// TwinCAT 3 PLC project tcp_client
// ProgramVersion: 3.1.4024.0
// libraries:
//   Tc2_Standard, * (Beckhoff Automation GmbH)
//   Tc2_System, * (Beckhoff Automation GmbH)
//   Tc2_TcpIp, * (Beckhoff Automation GmbH)
//   Tc3_Module, * (Beckhoff Automation GmbH)
// project tree:
//   GVLs/ SockParam.TcGVL
//   / PlcTask.TcTTO
//   POUs/libSocketClient/ E_SocketCommStateMachine.TcDUT, FB_SocketClientController.TcPOU, FB_MessageQueue.TcPOU, ITF_Receiver.TcIO, ITF_Sender.TcIO, ITF_TaskObserver.TcIO, ST_CommunicationMetaData.TcDUT, ST_CommandContainer.TcDUT
//   POUs/ MAIN.TcPOU
//   POUs/protocols/ FB_SocketClientProtocolBase.TcPOU
//   POUs/protocols/TestProtocol/ FB_TestProtocol.TcPOU, ST_ReceiveDataFormat.TcDUT, ST_SendDataFormat.TcDUT
// real-time tasks:
//   TASK PlcTask: cycle T#10ms, priority 20, ADS port 350

CONFIGURATION tcp_client
    RESOURCE PLC ON TwinCAT3
        TASK PlcTask(INTERVAL := T#10ms, PRIORITY := 20);
        PROGRAM MAIN WITH PlcTask : MAIN;
    END_RESOURCE
END_CONFIGURATION

// ---- POUs/libSocketClient/E_SocketCommStateMachine.TcDUT
{attribute 'qualified_only'}
{attribute 'strict'}
TYPE E_SocketCommStateMachine :
(
	init := 0,
	connect,
	idle,
	send,
	receive,
	disconnect,
	done
);
END_TYPE

// ---- POUs/libSocketClient/ST_CommunicationMetaData.TcDUT
TYPE ST_CommunicationMetaData :
STRUCT
	cbLen	: UDINT;
	pData	: PVOID;
END_STRUCT
END_TYPE

// ---- POUs/libSocketClient/ST_CommandContainer.TcDUT
TYPE ST_CommandContainer :
STRUCT
	sender : ITF_Sender;
	receiver : ITF_receiver;
END_STRUCT
END_TYPE

// ---- POUs/protocols/TestProtocol/ST_ReceiveDataFormat.TcDUT
{attribute 'pack_mode' := '1'}
TYPE ST_ReceiveDataFormat :
STRUCT
   command        : STRING(4);
   seq_number    : ULINT;
   value        : STRING(10240);
END_STRUCT
END_TYPE

// ---- POUs/protocols/TestProtocol/ST_SendDataFormat.TcDUT
{attribute 'pack_mode' := '1'}
TYPE ST_SendDataFormat :
STRUCT
   command        : STRING(4);
   seq_number    : ULINT;
   value        : ULINT;
END_STRUCT
END_TYPE

// ---- GVLs/SockParam.TcGVL
{attribute 'qualified_only'}
VAR_GLOBAL CONSTANT
	MAX_MESSAGE_SIZE : UDINT := 2048;	// 受信処理バッファ最大サイズ
	RECEIVE_BUFFER_SIZE	: UDINT := 20480; // 受信メッセージの組立先のバッファサイズ
END_VAR

// ---- POUs/libSocketClient/ITF_Receiver.TcIO
INTERFACE ITF_Receiver EXTENDS __System.IQueryInterface

METHOD flush : BOOL
VAR_INPUT
END_VAR
END_METHOD

METHOD Parse : BOOL
VAR_INPUT
END_VAR
END_METHOD

PROPERTY received : BOOL
GET
END_GET
END_PROPERTY

METHOD ResetBufferPointer : BOOL
VAR_INPUT
END_VAR
END_METHOD

METHOD SetReceivedData : BOOL
VAR_INPUT
	pData	: PVOID;
	cbLen	: UDINT;
END_VAR
END_METHOD

END_INTERFACE

// ---- POUs/libSocketClient/ITF_Sender.TcIO
INTERFACE ITF_Sender EXTENDS __System.IQueryInterface

PROPERTY SendData : ST_CommunicationMetaData
GET
END_GET
END_PROPERTY

END_INTERFACE

// ---- POUs/libSocketClient/ITF_TaskObserver.TcIO
INTERFACE ITF_TaskObserver EXTENDS __System.IQueryInterface

PROPERTY activity : E_SocketCommStateMachine
GET
END_GET
SET
END_SET
END_PROPERTY

PROPERTY complete : BOOL
GET
END_GET
SET
END_SET
END_PROPERTY

PROPERTY error : BOOL
GET
END_GET
SET
END_SET
END_PROPERTY

PROPERTY error_id : UDINT
GET
END_GET
SET
END_SET
END_PROPERTY

END_INTERFACE

// ---- POUs/MAIN.TcPOU
PROGRAM MAIN
VAR
	protcol : FB_TestProtocol;
	controller : FB_SocketClientController;
	connect : BOOL;
	handle : T_HSOCKET;
	
	// Command execution
	command_interval_timer : TON := (PT := T#1S);
	rand : DRAND;
	busy : BOOL;
	// Receive data
	receive_data : REFERENCE TO ST_ReceiveDataFormat;	
	
END_VAR

IF connect THEN
	handle := controller.connect('127.0.0.1', 9998);
ELSE
	controller.disconnect();
	busy := FALSE;
END_IF

IF handle.handle <> 0 THEN
	command_interval_timer(IN := NOT command_interval_timer.Q);
	IF command_interval_timer.Q AND NOT busy THEN
		rand(Seed := 1);
		protcol.send_data.command := 'SEND';
		protcol.send_data.seq_number := protcol.send_data.seq_number + 1;
		protcol.send_data.value := TO_ULINT(rand.Num * 100000);
		controller.queue.put(protcol, protcol);
		busy := TRUE;
	END_IF
	IF busy AND protcol.complete THEN
		receive_data REF= protcol.receive_data;
		busy := FALSE;
	END_IF
END_IF

controller();

END_PROGRAM

// ---- POUs/protocols/TestProtocol/FB_TestProtocol.TcPOU

FUNCTION_BLOCK FB_TestProtocol EXTENDS FB_SocketClientProtocolBase
VAR_INPUT
	send_data : ST_SendDataFormat;
END_VAR
VAR_OUTPUT
	receive_data : ST_ReceiveDataFormat;
END_VAR
VAR
END_VAR

METHOD Parse : BOOL
IF SIZEOF(receive_data) = MEMCPY(ADR(receive_data), ADR(SUPER^.receive_data_buffer), SIZEOF(receive_data)) THEN
	Parse := TRUE;
END_IF
END_METHOD

PROPERTY received : BOOL
GET
VAR
	specified_size : UDINT;
END_VAR
specified_size := SIZEOF(receive_data);
received := SUPER^.receive_data_size = specified_size;
END_GET
END_PROPERTY

PROPERTY SendData : ST_CommunicationMetaData
GET
SendData.cbLen := SIZEOF(send_data);
SendData.pData := ADR(send_data);
END_GET
END_PROPERTY

END_FUNCTION_BLOCK

// ---- POUs/protocols/FB_SocketClientProtocolBase.TcPOU
FUNCTION_BLOCK ABSTRACT FB_SocketClientProtocolBase IMPLEMENTS ITF_Sender, ITF_Receiver, ITF_TaskObserver
VAR CONSTANT
	MAX_NUM_OF_REQUEST_SECTIONS : UINT := 16;
END_VAR
VAR_OUTPUT
	//ParsedStructVariable : ST_********;
END_VAR
VAR	
	expected_receive_size_min : UDINT := 1; 
	expected_receive_size_max : UDINT := 1024; 
	receive_data_buffer	: ARRAY [0..SockParam.RECEIVE_BUFFER_SIZE - 1] OF BYTE;
	receive_data_size	: UDINT;
	_activity : E_SocketCommStateMachine;
	_error		: BOOL;
	_complete	: BOOL;
	_error_id	: UDINT;
END_VAR

PROPERTY activity : E_SocketCommStateMachine
GET
activity := _activity;
END_GET
SET
_activity := activity;
END_SET
END_PROPERTY

PROPERTY complete : BOOL
GET
complete := _complete;
END_GET
SET
_complete := complete;
END_SET
END_PROPERTY

PROPERTY error : BOOL
GET
error := _error;
END_GET
SET
_error := error;
END_SET
END_PROPERTY

PROPERTY error_id : UDINT
GET
error_id := _error_id;
END_GET
SET
_error_id := error_id;
END_SET
END_PROPERTY

METHOD FB_init : BOOL
VAR_INPUT
	bInitRetains : BOOL; // if TRUE, the retain variables are initialized (warm start / cold start)
	bInCopyCode : BOOL;  // if TRUE, the instance afterwards gets moved into the copy code (online change)
END_VAR
THIS^.flush();
END_METHOD

METHOD flush : BOOL
receive_data_size := 0;
END_METHOD

METHOD Parse : BOOL
END_METHOD

PROPERTY received : BOOL
GET
END_GET
END_PROPERTY

METHOD ResetBufferPointer : BOOL
receive_data_size := 0;
END_METHOD

PROPERTY SendData : ST_CommunicationMetaData
GET
END_GET
END_PROPERTY

METHOD SetReceivedData : BOOL
VAR_INPUT
	pData	: PVOID;
	cbLen	: UDINT;
END_VAR
VAR
	i : UDINT;
END_VAR
IF pData = 0 OR cbLen = 0 THEN
	RETURN;
END_IF

MEMCPY(ADR(receive_data_buffer) + receive_data_size, pData, cbLen);
receive_data_size := receive_data_size + cbLen;
SetReceivedData := TRUE;
END_METHOD

END_FUNCTION_BLOCK

// ---- POUs/libSocketClient/FB_SocketClientController.TcPOU
FUNCTION_BLOCK FB_SocketClientController
VAR_INPUT
	bConnect        : BOOL;
END_VAR

VAR_OUTPUT
	bError			: BOOL;
	bBusy			: BOOL;
	nErrStep		: E_SocketCommStateMachine;
	nErrId			: UDINT;	
END_VAR

VAR
	receive_data_buffer : ARRAY[0..SockParam.MAX_MESSAGE_SIZE - 1] OF BYTE;
	
	_command_queue	: FB_MessageQueue;
	_command : REFERENCE TO ST_CommandContainer;
	
	// Tcp
	fbConnect		: FB_SocketConnect;
	fbClose			: FB_SocketClose;
	_sRemoteHost	: T_IPv4Addr;
	fbSend			: FB_SocketSend;
	fbReceive		: FB_SocketReceive;
	nState			:	E_SocketCommStateMachine;
	_sock_handle	: T_HSocket;
	bExecuteSend	: BOOL;
	eConnState		: E_SocketConnectionState;
	_nPort			: UDINT;
	_receiver		: ITF_Receiver;
	_sender			: ITF_Sender;
	_observer		: ITF_TaskObserver;
	send_data 		: ST_CommunicationMetaData;	
	_length_of_receive_data		: UDINT;
END_VAR

CASE nState OF
E_SocketCommStateMachine.init: 
	IF bConnect THEN
		initComms();
		bError := FALSE;
		nErrId	:= 0;
		nState := E_SocketCommStateMachine.connect;
	END_IF
E_SocketCommStateMachine.connect:
	fbConnect(													// Open connection to server
			sSrvNetId:= '', 
			sRemoteHost:= _sRemoteHost, 
			nRemotePort:= _nPort, 
			bExecute:= TRUE, 
			tTimeout:= T#4S, 
			bBusy=> , 
			bError=> bError, 
			hSocket=> _sock_handle);

	IF _sock_handle.handle <> 0 AND NOT (fbConnect.bBusy) THEN			// Handle is created
		fbConnect(bExecute := FALSE);
		nState := E_SocketCommStateMachine.idle;
	ELSIF fbConnect.bError THEN
		bError := fbConnect.bError;
		nErrId := fbConnect.nErrId;
		nErrStep := nState;
		nState := E_SocketCommStateMachine.done;
	END_IF
E_SocketCommStateMachine.idle: // Wait command ready event

	// コマンドキューデータが有れば取り出して _command 参照変数にコマンド構造体をセット。
	// コマンド構造体はITF_Sender, ITF_Receiverのインターフェースを格納。
	// タイムアウト等でサーバ側から切断された場合、fbSend()でエラーになり、Step0に戻る。
	// この後再接続してコマンドを再実行した場合、キューから取り出さずそのままコマンド実行する。
	// _cmmandはシーケンスが正常終了した際に無効な参照値を書き込むため、
	// この場合に限りキューからコマンドを取り出す条件としている。
	IF NOT __ISVALIDREF(_command) AND _command_queue.usage > 0 THEN
		_command REF= _command_queue.get(); // キューから取り出したコマンドをセットする。
	END_IF
	
	IF __ISVALIDREF(_command) THEN
		_sender := _command.sender;
		_receiver := _command.receiver;
		IF NOT __QUERYINTERFACE(_receiver, _observer) THEN
			IF NOT __QUERYINTERFACE(_sender, _observer) THEN
				_observer := 0;
			END_IF
		END_IF
		IF _observer <> 0 THEN
			_observer.complete := FALSE;
		END_IF
		_receiver.flush();
		fbSend(bExecute := FALSE);
		send_data := _sender.SendData;
		_receiver.ResetBufferPointer();
		bBusy := TRUE;
		nState := E_SocketCommStateMachine.send;
	END_IF
	
E_SocketCommStateMachine.send: // Send command
	fbSend(
		sSrvNetId:= '', 
		hSocket:= _sock_handle, 
		cbLen:= send_data.cbLen, 
		pSrc:= send_data.pData, 
		bExecute:= TRUE,
		tTimeout:= T#100MS, 
		bBusy=> bBusy);
	
	IF NOT fbSend.bBusy THEN									// Check cyclically for new data
			nState := E_SocketCommStateMachine.receive;
	END_IF
		
	//ReceiveMessage();
	IF fbSend.bError THEN							// Close connection in case of error or manual communication stop
		bError := fbSend.bError;
		nErrId := fbSend.nErrId;
		nErrStep := nState;
		nState := E_SocketCommStateMachine.disconnect;
	END_IF

E_SocketCommStateMachine.receive: //Receive
	fbSend(bExecute := FALSE);
	
	fbReceive(													// ReceiveData
		sSrvNetId:= '', 
		hSocket:= _sock_handle, 
		cbLen:= SIZEOF(receive_data_buffer), 
		pDest:=  ADR(receive_data_buffer), 
		bExecute:= true, 
		tTimeout:= T#100MS, 
		bBusy=> bBusy, 
		nRecBytes=> _length_of_receive_data);
	IF NOT fbReceive.bBusy THEN									// Check cyclically for new data
		fbReceive(bExecute := FALSE);
		IF fbReceive.bError THEN							// Close connection in case of error or manual communication stop
			bError := fbReceive.bError;
			nErrId := fbReceive.nErrId;
			nErrStep := nState;
			nState := E_SocketCommStateMachine.disconnect;
		ELSE
			_receiver.SetReceivedData(
				pData := ADR(receive_data_buffer),
				cbLen := _length_of_receive_data
			);
			IF _receiver.received THEN
				_receiver.Parse();
				bBusy := FALSE;
				_command REF= 0;	// 正常終了したらコマンド参照変数に無効値を書き込む
				_sender := 0;
				_receiver := 0;
				IF _observer <> 0 THEN
					_observer.complete := TRUE;
					_observer := 0;
				END_IF
				nState := E_SocketCommStateMachine.idle;
			END_IF
		END_IF
	END_IF
E_SocketCommStateMachine.disconnect://Disconnecting
	fbClose(														// Close connection
			sSrvNetId:= '', 
			hSocket:= _sock_handle, 
			bExecute:= TRUE, 
			tTimeout:= T#4S, 
			);
			
	IF fbClose.bError THEN
		bError := fbClose.bError;
		nErrId := fbClose.nErrId;
		nErrStep := nState;
	END_IF

	IF NOT fbClose.bBusy THEN
		_sock_handle.handle := 0;
		nState := E_SocketCommStateMachine.init;
		bConnect := FALSE;
	END_IF
E_SocketCommStateMachine.done:
	bConnect := FALSE;
	nState := E_SocketCommStateMachine.init;
END_CASE

IF nState > E_SocketCommStateMachine.connect AND nState <> E_SocketCommStateMachine.done AND NOT bConnect THEN
	nState := E_SocketCommStateMachine.disconnect;
END_IF

IF _observer <> 0 THEN
	_observer.error := bError;
	_observer.error_id := nErrId;
	IF bError THEN
		_observer.activity := nErrStep;
	ELSE
		_observer.activity := nState;
	END_IF
END_IF

METHOD connect : Tc2_TcpIp.T_HSOCKET
VAR_INPUT
	sIPAddr	: T_IPv4Addr := '127.0.0.1';
	nPort	: UDINT := 8888;
END_VAR
THIS^._sRemoteHost  := sIPAddr;
THIS^._nPort := nPort;
bConnect := TRUE;
IF nState >= E_SocketCommStateMachine.idle THEN
	connect := _sock_handle;
ELSE
	connect.handle := 0;
END_IF
END_METHOD

METHOD disconnect : BOOL
VAR_INPUT
END_VAR
bConnect := FALSE;
END_METHOD

PROPERTY hSocketHandle : T_HSocket
GET
hSocketHandle := _sock_handle;
END_GET
SET
_sock_handle := hSocketHandle;
END_SET
END_PROPERTY

METHOD PRIVATE initComms : BOOL
VAR_INPUT
END_VAR
fbConnect(bExecute := FALSE); 
fbClose(bExecute := FALSE);
fbSend(bExecute := FALSE); 
fbReceive(bExecute := FALSE);
_command REF= 0;
_sender := 0;
_receiver := 0;
_observer := 0;
bBusy := FALSE;
bError := FALSE;
nErrId := 0;
initComms := TRUE;
END_METHOD

PROPERTY queue : REFERENCE TO FB_MessageQueue
GET
queue REF= _command_queue;
END_GET
END_PROPERTY

END_FUNCTION_BLOCK

// ---- POUs/libSocketClient/FB_MessageQueue.TcPOU
FUNCTION_BLOCK FB_MessageQueue
VAR CONSTANT
	COMMAND_QUEUE_BUFFER_SIZE :UDINT := 5;
END_VAR
VAR_OUTPUT
END_VAR
VAR
	_usage:	UDINT;
	_write_index : UDINT := 1;
	_read_index : UDINT := 1;
	_queue_size:	UDINT := COMMAND_QUEUE_BUFFER_SIZE;
	queue_buffer:	ARRAY [1..COMMAND_QUEUE_BUFFER_SIZE] OF ST_CommandContainer;
END_VAR

PROPERTY full : BOOL
GET
full :=  _usage >= COMMAND_QUEUE_BUFFER_SIZE;
END_GET
END_PROPERTY

METHOD get : REFERENCE TO ST_CommandContainer
VAR_INPUT
END_VAR
IF _usage = 0 THEN
	get REF= 0;
	RETURN;
END_IF

get REF= queue_buffer[_read_index];

_usage := _usage - 1;

IF COMMAND_QUEUE_BUFFER_SIZE > _read_index THEN
	_read_index := _read_index + 1;
ELSE
	_read_index := 1;
END_IF
END_METHOD

METHOD put : BOOL
VAR_INPUT
	sender : ITF_Sender;
	receiver : ITF_Receiver;
END_VAR
IF _usage >= COMMAND_QUEUE_BUFFER_SIZE THEN
	put := FALSE;
ELSE
	queue_buffer[_write_index].sender := sender;
	queue_buffer[_write_index].receiver := receiver;
	_usage := _usage + 1;
	IF COMMAND_QUEUE_BUFFER_SIZE > _write_index THEN
		_write_index := _write_index + 1;
	ELSE
		_write_index := 1;
	END_IF
	put := TRUE;
END_IF
END_METHOD

PROPERTY usage : UDINT
GET
usage := _usage;
END_GET
END_PROPERTY

END_FUNCTION_BLOCK
